// TIA Portal V18 export
DATA_BLOCK "Block_1_DB"   // DB2
VERSION : 0.1
// stored: AutoNumber true, InstanceOfName Block_1, InstanceOfType FB
"Block_1"
   // VAR_INPUT
   //    w1 : Bool;
   // END_VAR
   // VAR_OUTPUT
   //    w2 : Bool;
   // END_VAR
   // VAR
   //    IEC_Timer_0_Instance { S7_SetPoint := 'True'} : TON_TIME;
   // END_VAR
BEGIN
END_DATA_BLOCK
